INTERFACE ITF_AnalogSensor

PROPERTY Value : INT
GET
END_GET
END_PROPERTY

END_INTERFACE

(* stored: Version 1.1.0.1, ProductVersion 3.1.4024.9
   Itf ITF_AnalogSensor: Id {046937c7-7fca-4c6d-ba98-77d1fe003aff}
   Property Value: Id {31234351-ee15-4997-8056-e8bb4163cc3b}
   Get Get: Id {4b526d69-f2e7-4548-ab5c-d9240b4ab5dc} *)
